SUBAPPLICATION Uebung_010c3_sub_AX (* SoftKey_F1 auf DigitalOutput_Q1 mit GreenWhiteBackground mit Typed Subapp *)
  (* Standard: 61499-2; Description: Copyright (c) 2026 Meisterschulen am Ostbahnhof This program and the accompanying materials are made available under the terms of the Eclipse Public License 2.0 which is available at https://www.eclipse.org/legal/epl-2.0/ SPDX-License-Identifier: EPL-2.0 *)
  (* Version 1.0, 2026-01-15, Moritz Ortmeier, Meisterschulen am Ostbahnhof *)
  PACKAGE Uebungen;
  IMPORT isobus::UT::Q::const::IDs::ID_NULL;
  IMPORT logiBUS::io::DQ::logiBUS_DO;
  IMPORT logiBUS::io::DQ::logiBUS_DO_S;
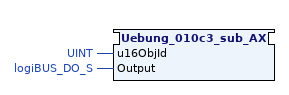
  VAR_INPUT
    u16ObjId : UINT := ID_NULL; (* Object ID *)
    Output : logiBUS::io::DQ::logiBUS_DO_S := logiBUS_DO::Invalid; (* Identify the Output Output_Q1..Q8 *)
  END_VAR
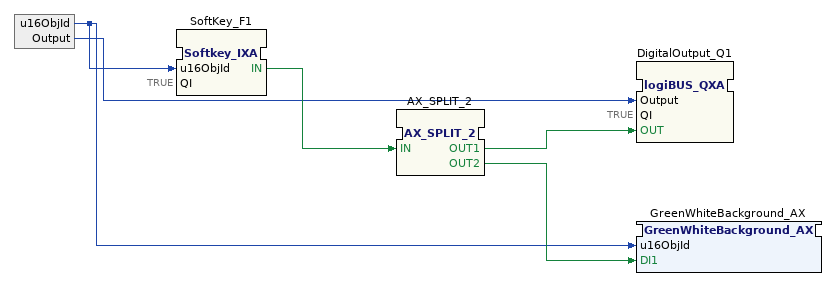
  FBS
    DigitalOutput_Q1 : logiBUS::io::DQ::logiBUS_QXA(QI := TRUE);
    SoftKey_F1 : isobus::UT::io::Softkey::Softkey_IXA(QI := TRUE);
    AX_SPLIT_2 : adapter::events::unidirectional::AX_SPLIT_2;
  END_FBS
  SUBAPPS
    GreenWhiteBackground_AX : MyLib::sys::GreenWhiteBackground_AX;
  END_SUBAPPS
  DATA_CONNECTIONS
    u16ObjId TO SoftKey_F1.u16ObjId;
    u16ObjId TO GreenWhiteBackground_AX.u16ObjId;
    Output TO DigitalOutput_Q1.Output;
  END_CONNECTIONS
  ADAPTER_CONNECTIONS
    SoftKey_F1.IN TO AX_SPLIT_2.IN;
    AX_SPLIT_2.OUT1 TO DigitalOutput_Q1.OUT;
    AX_SPLIT_2.OUT2 TO GreenWhiteBackground_AX.DI1;
  END_CONNECTIONS
END_SUBAPPLICATION
